// TIA Portal V20 export
VAR_GLOBAL   // PLC tag table "OutPut Equipment"
   q_xTableCheck_LampNG_p1 AT %Q5.0 : Bool;   // Output - indication lamp, NO good operation for table P1
   q_xTableCheck_LampOK_p1 AT %Q5.1 : Bool;   // Output - indication lamp, Ok operation for table P1
   q_xTableCheck_LampNG_p2 AT %Q5.2 : Bool;   // Output - indication lamp, NO good operation for table P2
   q_xTableCheck_LampOK_p2 AT %Q5.3 : Bool;   // Output - indication lamp, Ok operation for table P2
END_VAR
